TYPE ST_Cylinder_Command :
    STRUCT
        Extend  : BOOL;
        Retract : BOOL;
    END_STRUCT
END_TYPE

(* stored: Version 1.1.0.1, ProductVersion 3.1.4024.15
   DUT ST_Cylinder_Command: Id {da610787-8da4-0918-242c-6ff79d9b522a} *)
